{attribute 'GeneratedUsingTerminal: EK1960-0000-0021'}
{attribute addProperty BoxType "EK1960-0000-0021"}
{attribute addProperty Id "FSOEAT %I*FSOE_39DE0EE047"}
{attribute addProperty CRC "1823951946"}
{attribute addProperty Size "47"}
TYPE FSoE_Inputs_6CB74C4A :
STRUCT
	{attribute addProperty Name "FSOE"}
	FSOE AT %I* : FSOE_39DE0EE0;
END_STRUCT
END_TYPE

(* stored: Version 1.2.0.0, ProductVersion 3.1.4024.9
   DUT FSoE_Inputs_6CB74C4A: Id {af0bd136-aa22-4d36-bb3c-bd9ea7549176} *)
